{attribute 'linkalways'} 
{attribute 'no_explicit_call' := 'This FB is a CLASS and must be accessed using methods or properties'}
{attribute 'enable_dynamic_creation'}
FUNCTION_BLOCK _ETcVnReduceType EXTENDS EnumDatatypeBase
VAR
	localData : ETcVnReduceType;
	activeData : REFERENCE TO ETcVnReduceType;
	enumBaseDatatype : _DINT(localData);
END_VAR

METHOD PRIVATE AddLocalEnumeration
VAR_INPUT
	Enumeration : T_MAXSTRING;
	Value : ETcVnReduceType;
END_VAR
AddEnumeration(Enumeration, Value);
END_METHOD

PROPERTY PUBLIC Address : PVOID
GET
Address := ADR(activeData);
END_GET
END_PROPERTY

METHOD PUBLIC ClearReference
VAR_INPUT
END_VAR
activeData REF= localData;
SetBaseDatatypeReference();
END_METHOD

METHOD PUBLIC Clone : I_Datatype
VAR
    pClone : POINTER TO _ETcVnReduceType;
END_VAR
pClone := __NEW(_ETcVnReduceType(InitialValue := Value));
Clone := pClone^;
END_METHOD

METHOD FB_init : BOOL
VAR_INPUT
	bInitRetains : BOOL; // if TRUE, the retain variables are initialized (warm start / cold start)
	bInCopyCode : BOOL;  // if TRUE, the instance afterwards gets moved into the copy code (online change)
	InitialValue : ETcVnReduceType;
END_VAR
localData := InitialValue;
AddBaseDatatype(enumBaseDatatype);
ClearReference();

AddLocalEnumeration('TCVN_RT_REDUCE_SUM', ETcVnReduceType.TCVN_RT_REDUCE_SUM);
AddLocalEnumeration('TCVN_RT_REDUCE_AVG', ETcVnReduceType.TCVN_RT_REDUCE_AVG);
AddLocalEnumeration('TCVN_RT_REDUCE_MAX', ETcVnReduceType.TCVN_RT_REDUCE_MAX);
AddLocalEnumeration('TCVN_RT_REDUCE_MIN', ETcVnReduceType.TCVN_RT_REDUCE_MIN);
END_METHOD

PROPERTY PUBLIC Identifier : T_MAXSTRING
GET
Identifier := 'ETcVnReduceType';
END_GET
END_PROPERTY

METHOD IsEnumeratorValueEqual : BOOL
VAR_INPUT
	Enumerator : I_KeyValueForwardEnumerator;
END_VAR
VAR
	storedValue : ETcVnReduceType;
END_VAR
IF NOT Enumerator.TryGet(storedValue) THEN
	RETURN;
END_IF

IsEnumeratorValueEqual := storedValue = activeData;
END_METHOD

METHOD PUBLIC MakeReferenceTo
VAR_INPUT
	ReferenceTarget : REFERENCE TO ETcVnReduceType;
END_VAR
activeData REF= ReferenceTarget;
SetBaseDatatypeReference();
END_METHOD

METHOD PROTECTED SetBaseDatatypeReference
VAR_INPUT
END_VAR
enumBaseDatatype.MakeReferenceTo(activeData);
END_METHOD

PROPERTY PUBLIC Size : UDINT
GET
Size := SIZEOF(activeData);
END_GET
END_PROPERTY

METHOD TryMakeReferenceTo : BOOL
VAR_INPUT
	Target : I_Datatype;
END_VAR
VAR
	pTargetData : POINTER TO ETcVnReduceType;
END_VAR
IF NOT IsEquivalentTo(Target) THEN
	RETURN;
END_IF

pTargetData := Target.Address;
activeData REF= pTargetData^;
SetBaseDatatypeReference();
TryMakeReferenceTo := TRUE;
END_METHOD

PROPERTY PUBLIC Value : ETcVnReduceType
GET
Value := activeData;
END_GET
SET
activeData := Value;
END_SET
END_PROPERTY

END_FUNCTION_BLOCK

(* stored: Version 1.1.0.1, ProductVersion 3.1.4024.15
   POU _ETcVnReduceType: Id {088b7d7c-59f3-0897-2d67-ba21c6f1f824}, SpecialFunc None
   Folder Core: Id {9d7f35fc-e181-08bf-1e69-71fa5f0cd8fb}
   Folder Protected: Id {85e46457-3957-0245-1e48-8f29fb7754e2}
   Folder Customize: Id {57037c45-008f-04d3-204a-9b20bde5e958}
   Folder Constructor: Id {aa5be6b3-033b-078b-1543-0f347fcb3279}
   Folder Private: Id {199589d9-9b97-0ac3-23b5-5b20aa1b50d6}
   Folder Protected: Id {dfb793d4-9a8d-0478-0d1b-a3be29f98a7e}
   Method AddLocalEnumeration: Id {fc3c6860-4072-0d5a-16f0-fef1b4db4909}
   Property Address: Id {e54d317f-0743-000f-3247-2616bf4286b4}
   Get Get: Id {553e5011-3ca7-044e-1c26-6e8e7ee61d35}
   Method ClearReference: Id {7abc10c2-c6e8-0ae0-11ec-6053d16d5992}
   Method Clone: Id {9e80086f-0519-0c38-036e-feff7b7ea9de}
   Method FB_init: Id {a728faec-f384-0abc-0e89-f8a4f614f210}
   Property Identifier: Id {77189ebe-c088-02a6-2d8e-a5ac6ac6b03a}
   Get Get: Id {1ab8922c-c71e-0217-1614-956cc8e057b0}
   Method IsEnumeratorValueEqual: Id {22882b35-ed6c-05d4-13c3-374497d3a61d}
   Method MakeReferenceTo: Id {b00f8a7c-a00f-0b74-1afd-a8d832419b02}
   Method SetBaseDatatypeReference: Id {ad8f743a-1ca0-0de7-1807-79565cc01542}
   Property Size: Id {6b818042-bf9f-0450-3b89-8fafbf50a35a}
   Get Get: Id {8329443e-e974-00b3-1993-0cd2877ace63}
   Method TryMakeReferenceTo: Id {7450873f-15ef-035d-3e82-525930b7bf79}
   Property Value: Id {03f3bed8-1d4f-0132-1962-26303c3733fc}
   Get Get: Id {d8b60931-6c17-0af9-37b5-85c70b6878c2}
   Set Set: Id {a0f312d0-219e-0b17-0045-e5eaf134bc16} *)
